SYSTEM Robot_client
  (* Version 1.0, 2025-07-16, felix *)
  APPLICATION Robot_clientApp
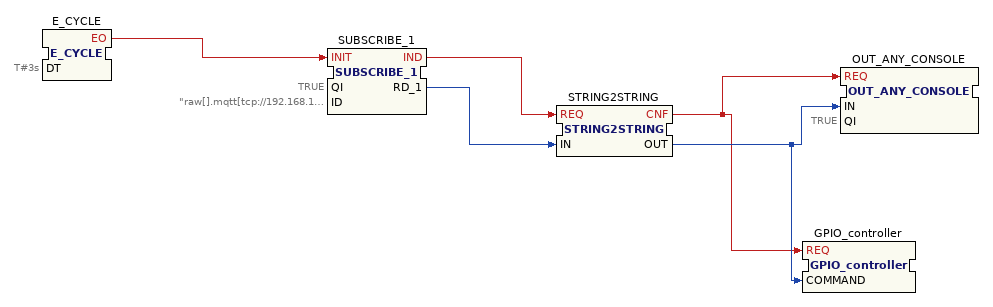
    FBS
      SUBSCRIBE_1 : SUBSCRIBE_1(QI := TRUE, ID := "raw[].mqtt[tcp://192.168.1.103:1883,forte,robot/gpio]");
      STRING2STRING : STRING2STRING;
      OUT_ANY_CONSOLE : OUT_ANY_CONSOLE(QI := TRUE);
      GPIO_controller : GPIO_controller;
      E_CYCLE : E_CYCLE(DT := T#3s);
    END_FBS
    EVENT_CONNECTIONS
      SUBSCRIBE_1.IND TO STRING2STRING.REQ;
      STRING2STRING.CNF TO OUT_ANY_CONSOLE.REQ;
      E_CYCLE.EO TO SUBSCRIBE_1.INIT;
      STRING2STRING.CNF TO GPIO_controller.REQ;
    END_CONNECTIONS
    DATA_CONNECTIONS
      SUBSCRIBE_1.RD_1 TO STRING2STRING.IN;
      STRING2STRING.OUT TO OUT_ANY_CONSOLE.IN;
      STRING2STRING.OUT TO GPIO_controller.COMMAND;
    END_CONNECTIONS
  END_APPLICATION
  DEVICE FORTE_PC : FORTE_PC(MGR_ID := "192.168.1.101:61499" (* Device manager socket ID *))
    {SET_ATTRIBUTE(Profile, HOLOBLOC)}
    RESOURCE EMB_RES : EMB_RES
      EVENT_CONNECTIONS
        START.COLD TO Robot_clientApp.E_CYCLE.START;
        START.WARM TO Robot_clientApp.E_CYCLE.START;
      END_CONNECTIONS
    END_RESOURCE
  END_DEVICE
  MAPPINGS
    Robot_clientApp.SUBSCRIBE_1 ON FORTE_PC.EMB_RES;
    Robot_clientApp.STRING2STRING ON FORTE_PC.EMB_RES;
    Robot_clientApp.OUT_ANY_CONSOLE ON FORTE_PC.EMB_RES;
    Robot_clientApp.GPIO_controller ON FORTE_PC.EMB_RES;
    Robot_clientApp.E_CYCLE ON FORTE_PC.EMB_RES;
  END_MAPPINGS
  SEGMENTS
    Ethernet : Ethernet;
  END_SEGMENTS
  LINKS
    FORTE_PC => Ethernet;
  END_LINKS
END_SYSTEM
